INTERFACE ITF_Control1_HMI_Init EXTENDS ITF_BaseControlElement, ITF_Control1_HMI_Connector

END_INTERFACE

(* stored: Version 1.1.0.1
   Itf ITF_Control1_HMI_Init: Id {b0fc800d-2a41-0aef-3282-732a4350c9fa} *)
